# EPICS substitutions: opcua-IOC-demoApp/Db/opcuaServer.substitutions
file "opcuaServerStatus.template"
{
  pattern { P, R, SESS, SUBS }
          { "$(PREF)", "$(REC=)", "$(SESSION)", "$(SUBSCRIPT)" }
}
